TYPE AxesManualTabs :
(
	TAB_POSITIONS := 0,
    TAB_JOYSTICK_AZIELE := 1,
    TAB_JOYSTICK_ROT := 2,
    TAB_OFFSETS_AZIELE := 3,
    TAB_OFFSETS_ALPHADELTA := 4,
    TAB_MOVEABSOLUTE := 5,
    TAB_MOVEVELOCITY  := 6
);
END_TYPE

(* stored: Version 1.1.0.1, ProductVersion 3.1.4019.2
   DUT AxesManualTabs: Id {a676ea36-0b8a-45ed-a02d-b67173e03fae} *)
